(* CODESYS project FU_CheckNumber.xml

Project tree, tasks and I/O mapping:
  function FU_CheckNumber [ST]
*)

// FU_CheckNumber
//This function checks if a string only contains numbers, dot (.) and dash (-) are also permitted as they are required for some numbers
//Returns true if string only contains numbers
// |**Version**|**Author**| **Date** |**Changes**
// | 1         | NSN      | 10-12-18 | Creation
FUNCTION FU_CheckNumber : BOOL
VAR_INPUT
	str			:STRING(255);	//String
END_VAR

FU_CheckNumber		:=		FU_CheckNumberBI(str:=str);

END_FUNCTION
